// TIA Portal V17 export
// export: Created 2022-06-21T13:51:02.2858297Z, ExportSetting WithDefaults, DisplayName Totally Integrated Automation Portal, DisplayVersion V17, DisplayName TIA Portal Openness, DisplayVersion V17, DisplayName TIA Portal Version Control Interface, DisplayVersion V17, DisplayName STEP 7 Professional, DisplayVersion V17, DisplayName STEP 7 Safety, DisplayVersion V17, DisplayName WinCC Advanced, DisplayVersion V17
VAR_GLOBAL   // PLC tag table "STEP7 classic symbols"
   P_AI_ARM2_INBOARD_ANGLE AT %IW512 : Word;
   P_AI_ARM2_OUTBOARD_ANGLE AT %IW514 : Word;
   P_AI_ARM2_SLEWING_ANGLE AT %IW516 : Word;
   I_PMS_AL_Z_TEST_KSW AT %I0.1 : Bool;
   I_PMS_ON_KSW AT %I0.0 : Bool;
   O_ARM1_2ND_ALARM_PMS_PLC AT %Q61.2 : Bool;
   O_ARM1_PRE_ALARM_PMS_PLC AT %Q61.0 : Bool;
   O_ARM2_1ST_ALARM_PMS_PLC AT %Q62.1 : Bool;
   O_ARM2_2ND_ALARM_PMS_PLC AT %Q62.2 : Bool;
   O_ARM2_PRE_ALARM_PMS_PLC AT %Q62.0 : Bool;
   O_CPU_PMS_FAULT_PLC AT %Q60.3 : Bool;
   O_PMS_ON_PMS AT %Q60.7 : Bool;
   O_SENSORS_FAILURE_PMS AT %Q60.6 : Bool;
   O_UPDATE_PREALARM AT %Q60.5 : Bool;
   O_1ST_ALARM_PMS_PLC AT %Q60.1 : Bool;
   O_2ND_ALARM_PMS_PLC AT %Q60.2 : Bool;
   O_ALARM_ZONE_TES_PLC AT %Q60.0 : Bool;
   O_ARM1_1ST_ALARM_PMS_PLC AT %Q61.1 : Bool;
   BM900 AT %MW102 : Int;   // = 3
   sim_mla3 AT %M200.2 : Bool;
   sim_mla4 AT %M200.3 : Bool;
   sim_mla5 AT %M200.4 : Bool;
   sim_mla6 AT %M200.5 : Bool;
   sim_mla7 AT %M200.6 : Bool;
   sim_mla8 AT %M200.7 : Bool;
   sim_mla9 AT %M201.0 : Bool;
   sim_x1 AT %MW250 : Int;
   sim_x10 AT %MW304 : Int;
   sim_x2 AT %MW256 : Int;
   sim_x3 AT %MW262 : Int;
   sim_x4 AT %MW268 : Int;
   sim_x5 AT %MW274 : Int;
   sim_x6 AT %MW280 : Int;
   sim_x7 AT %MW286 : Int;
   sim_x8 AT %MW292 : Int;
   PUMP1 AT %MW32 : Int;   // = 1
   PUMP2 AT %MW34 : Int;   // = 2
   sim_z5 AT %MW278 : Int;
   sim_z6 AT %MW284 : Int;
   sim_z7 AT %MW290 : Int;
   sim_z8 AT %MW296 : Int;
   sim_z9 AT %MW302 : Int;
   sim_angle_tol AT %MD374 : Real;
   sim_dist_min_tol AT %MD378 : Real;
   sim_dist_tol AT %MD370 : Real;
   sim_mla1 AT %M200.0 : Bool;
   sim_mla10 AT %M201.1 : Bool;
   sim_mla2 AT %M200.1 : Bool;
   CP341_2_ERROR_NR AT %MW192 : Word;
   CP341_2_NDR AT %M190.2 : Bool;
   CP341_2_START AT %M190.0 : Bool;
   CP341_2_START_ERROR AT %M190.4 : Bool;
   CP341_2_START_FM AT %M190.1 : Bool;
   CP341_2_START_OK AT %M190.3 : Bool;
   Write_BM900 AT %MW96 : Int;   // = 6
   sim_y1 AT %MW252 : Int;
   sim_y10 AT %MW306 : Int;
   sim_y2 AT %MW258 : Int;
   sim_y3 AT %MW264 : Int;
   sim_y4 AT %MW270 : Int;
   sim_y5 AT %MW276 : Int;
   sim_y6 AT %MW282 : Int;
   sim_y7 AT %MW288 : Int;
   sim_y8 AT %MW294 : Int;
   sim_y9 AT %MW300 : Int;
   sim_z1 AT %MW254 : Int;
   sim_z10 AT %MW308 : Int;
   sim_z2 AT %MW260 : Int;
   sim_z3 AT %MW266 : Int;
   sim_z4 AT %MW272 : Int;
   FPI AT %MW100 : Int;   // = 2
   MLA8 AT %MW50 : Int;   // = 8
   MLA9 AT %MW52 : Int;   // = 9
   MLAMAX AT %MW58 : Int;   // Bigest number of an MLA in service. ie. 6 if MLA 7 to 10 don't exist.
   MLAMIN AT %MW56 : Int;   // Smallest number of an MLA in service. ie. 2 if the MLA 1 is not in service.
   MLA_SELECTED_NUM AT %MW30 : Int;   // 0: no MLA selected - 1: MLA n°1 selected - 2: MLA n°2 selected - ...
   M90 AT %MW98 : Int;   // = 1
   CP341_1_NDR AT %M180.2 : Bool;
   CP341_1_START AT %M180.0 : Bool;
   CP341_1_START_ERROR AT %M180.4 : Bool;
   CP341_1_START_FM AT %M180.1 : Bool;
   CP341_1_START_OK AT %M180.3 : Bool;
   CP341_2_ERROR_INFO AT %MW194 : Word;
   test_num AT %MW382 : Int;   // used for test in correlation
   x AT %MW80 : Int;   // = 1
   y AT %MW82 : Int;   // = 2
   z AT %MW84 : Int;   // = 3
   sim_x9 AT %MW298 : Int;
   MLA1 AT %MW36 : Int;   // = 1
   MLA10 AT %MW54 : Int;   // = 10
   MLA2 AT %MW38 : Int;   // = 2
   MLA3 AT %MW40 : Int;   // = 3
   MLA4 AT %MW42 : Int;   // = 4
   MLA5 AT %MW44 : Int;   // = 5
   MLA6 AT %MW46 : Int;   // = 6
   MLA7 AT %MW48 : Int;   // = 7
   Write_FPI AT %MW92 : Int;   // = 4
   Write_M90 AT %MW88 : Int;   // = 2
   CP341_1_ERROR_INFO AT %MW184 : Word;
   CP341_1_ERROR_NR AT %MW182 : Word;
   Read_BM900 AT %MW94 : Int;   // = 5
   Read_FPI AT %MW90 : Int;   // = 3
   Read_M90 AT %MW86 : Int;   // = 1
   LG_RECV AT %MW470 : Int;
   LG_RECV2 AT %MW472 : Int;
   LG_SEND AT %MW474 : Word;
   Arm1_Prealarm_Delay AT %T31 : Timer;
   Arm2_Prealarm_Delay AT %T32 : Timer;
   Arm3_Prealarm_Delay AT %T33 : Timer;
   Arm4_Prealarm_Delay AT %T34 : Timer;
   Arm5_Prealarm_Delay AT %T35 : Timer;
   Arm6_Prealarm_Delay AT %T36 : Timer;
   Arm7_Prealarm_Delay AT %T37 : Timer;
   Arm8_Prealarm_Delay AT %T38 : Timer;
   Arm9_Prealarm_Delay AT %T39 : Timer;
   Tempo_mla_9_corr_ok AT %T9 : Timer;   // When MLA 9 correlation is again ok, tempo before MLA 9 ok declaration
   CP341_2_MODBUS_DELAY AT %T81 : Timer;
   Start_Pogram_Timer AT %T20 : Timer;
   TEMPO_PUMP_ON AT %T0 : Timer;   // Maximum time to keep the selected pump On without any hydraulic action
   Tempo_mla_10_corr_ok AT %T10 : Timer;   // When MLA 10 correlation is again ok, tempo before MLA 10 ok declaration
   Tempo_mla_1_corr_ok AT %T1 : Timer;   // When MLA 1 correlation is again ok, tempo before MLA 1 ok declaration
   Tempo_mla_2_corr_ok AT %T2 : Timer;   // When MLA 2 correlation is again ok, tempo before MLA 2 ok declaration
   Tempo_mla_3_corr_ok AT %T3 : Timer;   // When MLA 3 correlation is again ok, tempo before MLA 3 ok declaration
   Tempo_mla_4_corr_ok AT %T4 : Timer;   // When MLA 4 correlation is again ok, tempo before MLA 4 ok declaration
   Tempo_mla_5_corr_ok AT %T5 : Timer;   // When MLA 5 correlation is again ok, tempo before MLA 5 ok declaration
   Tempo_mla_6_corr_ok AT %T6 : Timer;   // When MLA 6 correlation is again ok, tempo before MLA 6 ok declaration
   Tempo_mla_7_corr_ok AT %T7 : Timer;   // When MLA 7 correlation is again ok, tempo before MLA 7 ok declaration
   Tempo_mla_8_corr_ok AT %T8 : Timer;   // When MLA 8 correlation is again ok, tempo before MLA 8 ok declaration
   Fin_Calage_Delay AT %T120 : Timer;
   Arm10_Prealarm_Delay AT %T40 : Timer;
   Sensor_Failure_Delay AT %T21 : Timer;
   WATCHDOG_PLC AT %MD2 : DWord;
   Cycle_Time AT %M6.0 : LReal;
   Memo_Last_Cycle AT %M14.0 : LReal;
   Simu_on AT %M22.0 : Bool;
   raz AT %M22.1 : Bool;
   SP_SLEW AT %M60.0 : LReal;
   SP_INBOARD AT %M68.0 : LReal;
   SP_OUTBOARD AT %M104.0 : LReal;
   "V1(k)" AT %M112.0 : LReal;
   "V2(k)" AT %M120.0 : LReal;
   "V3(k)" AT %M128.0 : LReal;
   POS_SLEW AT %M136.0 : LReal;
   POS_INB AT %M144.0 : LReal;
   POS_OUTB AT %M152.0 : LReal;
   "φ(k)" AT %M160.0 : LReal;
   "α(k)" AT %M168.0 : LReal;
   "β(k)" AT %M204.0 : LReal;
   "θ2(k)" AT %M212.0 : LReal;
   "θ4(k)" AT %M220.0 : LReal;
   "θ6(k)" AT %M228.0 : LReal;
   "X(k)" AT %M236.0 : LReal;
   "Y(k)" AT %M310.0 : LReal;
   "Z(k)" AT %M318.0 : LReal;
   "θ2(k+1)" AT %M326.0 : LReal;
   "θ4(k+1)" AT %M334.0 : LReal;
   "θ6(k+1)" AT %M342.0 : LReal;
   "X(k+1)" AT %M350.0 : LReal;
   "Y(k+1)" AT %M358.0 : LReal;
   "Z(k+1)" AT %M384.0 : LReal;
   Easy_ON AT %M22.2 : Bool;
   A3_Cbr AT %M392.0 : LReal;
   A3_Cin AT %M400.0 : LReal;
   A3_Cout AT %M408.0 : LReal;
   "A2_φ(t)_simulé" AT %M416.0 : LReal;
   "A2_α(t)_simulé" AT %M424.0 : LReal;
   "A2_β(t)_simulé" AT %M432.0 : LReal;
   "AO_EV_SLEWING_%" AT %M440.0 : LReal;
   "AO_EV_INBOARD_%" AT %M448.0 : LReal;
   "AO_EV_OUTBOARD_%" AT %M456.0 : LReal;
   TEMP_FM_1HZ AT %M22.3 : Bool;
   LG_RECV3 AT %MW24 : Word;
   LG_RECV4 AT %MW26 : Word;
   LG_SEND_EASY AT %MW28 : Word;
   No_Motions AT %M22.4 : Bool;
   ZERO_LR AT %M476.0 : LReal;
   IN_TEST_LR AT %M484.0 : LReal;
   "A3_φ(t)_simulé" AT %M492.0 : LReal;
   "A3_α(t)_simulé" AT %M500.0 : LReal;
   "A3_β(t)_simulé" AT %M508.0 : LReal;
   A2_Cbr AT %M516.0 : LReal;
   A2_Cin AT %M524.0 : LReal;
   A2_Cout AT %M532.0 : LReal;
   A4_Cbr AT %M540.0 : LReal;
   A4_Cin AT %M548.0 : LReal;
   A4_Cout AT %M556.0 : LReal;
   "A4_β(t)_simulé" AT %M564.0 : LReal;
   "A4_α(t)_simulé" AT %M572.0 : LReal;
   "A4_φ(t)_simulé" AT %M580.0 : LReal;
   "A5_β(t)_simulé" AT %M588.0 : LReal;
   "A5_α(t)_simulé" AT %M596.0 : LReal;
   "A5_φ(t)_simulé" AT %M604.0 : LReal;
   A5_Cout AT %M612.0 : LReal;
   A5_Cin AT %M620.0 : LReal;
   A5_Cbr AT %M628.0 : LReal;
   Cbr AT %M636.0 : LReal;
   Cin AT %M644.0 : LReal;
   Cout AT %M652.0 : LReal;
END_VAR
